% RSLogix 500 project BIN SCRUBBER WITH ROTATING CRADEL TEST_BAK024.RSS, saved by version 11.00.00.00 %
PROJECT "UNTITLED"    % processor: MicroLogix 1200 %

PROGRAM FILES
  LAD 2   4 rungs

DATA FILES
  O0 OUTPUT  4 elements
  I1 INPUT  4 elements
  S2 STATUS  66 elements
  B3 BINARY  2 elements
  T4 TIMER  4 elements
  C5 COUNTER  1 elements
  R6 CONTROL  1 elements
  N7 INTEGER  1 elements
  F8 FLOAT  1 elements

LADDER 2
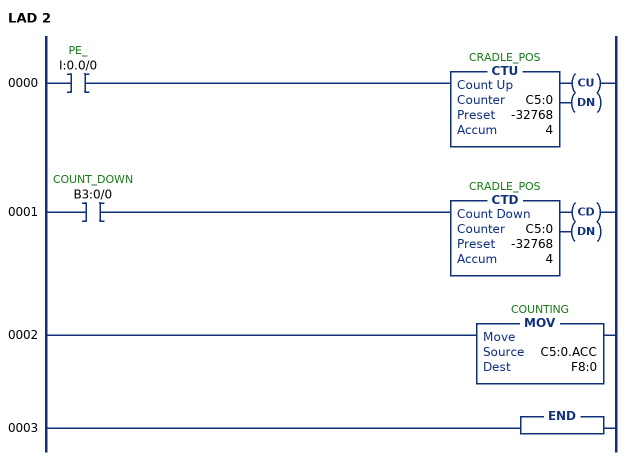
% Rung: 0 %
SOR XIC I:0.0/0 CTU C5:0 -32768 4 EOR
%   I:0.0/0  PE_ %
%   C5:0  CRADLE_POS %
% Rung: 1 %
SOR XIC B3:0/0 CTD C5:0 -32768 4 EOR
%   B3:0/0  COUNT_DOWN %
%   C5:0  CRADLE_POS %
% Rung: 2 %
SOR MOV C5:0.ACC F8:0 EOR
%   C5:0  CRADLE_POS %
%   F8:0  COUNTING %
% Rung: 3 %
SOR END EOR

OTHER DOCUMENTED ADDRESSES
  B3:0/1  FWD
  B3:0/2  CRADLE_DN
  B3:0/4  OSR_FWD
  B3:0/6  OSR_CCW
  B3:0/7  REV
  B3:0/9  OSF_PE
  B3:0/11  IN_POSITION_LIGHT
  B3:0/12  FWD_PE_IN_POS
  B3:0/13  REV_PE_IN_POS
  B3:0/14  STORAGE
  B3:0/15  ONS_RISING_RES_REV
  B3:1/0  STORAGE_BIT
  B3:1/1  ONS_RESET_FWD
  B3:3  OSR_STORAGE
  B3:4  FWD_COUNT
  B3:5  OSR_STORAGE_2
  B3:6  OSR_REVERSE
  B3:15  ONS_RESET_REV
  C5  
  CT5  
  CT54:5  COUNTER
  I:0.0/1  CLOCKWISE_FWD
  I:0.0/2  CRADLE_DOWN
  N7:0  LOOKUP
  O:0.0/0  FWD_MOTOR
  O:0.0/1  REV_MOTOR
  T4:0  ONESHOT_POS_CH_DISAB
  T4:1  PE_DEBOUNCE
  T4:2  PE_OFF_DEBOUNCE
  T4:3/TT  ONESHOT_POS_CH_DISA

DATA TABLE (non-zero values as saved)
DATA B3
% B3:0 % 0X0101 0X0000
DATA T4
% .PRE .ACC %
% T4:0 % 100 0
% T4:1 % 15 0
% T4:2 % 20 20
% T4:3 % 100 0
DATA C5
% .PRE .ACC %
% C5:0 % -32768 4
DATA N7
% N7:0 % 1
DATA F8
% F8:0 % 4
